  [768] = "0.00,0.00,0.00,90.00,0.00,90.00,0,"
  [769] = "0.00,0.00,0.00,90.00,0.00,90.00,0,"
  [770] = "0.00,0.00,0.00,90.00,0.00,90.00,0,"
  [771] = "0.00,0.00,0.00,90.00,0.00,90.00,1,"
  [772] = "0.00,0.00,0.00,90.00,0.00,90.00,0,"
  [773] = "0.00,0.00,0.00,90.00,0.00,90.00,0,"
  [774] = "0.00,0.00,0.00,90.00,0.00,90.00,0,"
  [775] = "0.00,0.00,0.00,90.00,0.00,90.00,1,"
  [776] = "0.00,0.00,0.00,90.00,0.00,90.00,0,"
  [777] = "0.00,0.00,0.00,90.00,0.00,90.00,0,"
  [778] = "0.00,0.00,0.00,90.00,0.00,90.00,0,"
  [779] = "0.00,0.00,0.00,90.00,0.00,90.00,1,"
  [780] = "0.00,0.00,0.00,90.00,0.00,90.00,0,"
  [781] = "0.00,0.00,0.00,90.00,0.00,90.00,0,"
  [782] = "0.00,0.00,0.00,90.00,0.00,90.00,0,"
  [783] = "0.00,0.00,0.00,90.00,0.00,90.00,1,"
  [784] = "0.00,0.00,0.00,90.00,0.00,90.00,0,"
  [785] = "0.00,0.00,0.00,90.00,0.00,90.00,0,"
  [786] = "0.00,0.00,0.00,90.00,0.00,90.00,0,"
  [787] = "0.00,0.00,0.00,90.00,0.00,90.00,1,"
  [788] = "0.00,0.00,0.00,90.00,0.00,90.00,0,"
  [789] = "0.00,0.00,0.00,90.00,0.00,90.00,0,"
  [790] = "0.00,0.00,0.00,90.00,0.00,90.00,0,"
  [791] = "0.00,0.00,0.00,90.00,0.00,90.00,1,"
  [792] = "0.00,0.00,0.00,90.00,0.00,90.00,0,"
  [793] = "0.00,0.00,0.00,90.00,0.00,90.00,0,"
  [794] = "0.00,0.00,0.00,90.00,0.00,90.00,0,"
  [795] = "0.00,0.00,0.00,90.00,0.00,90.00,1,"
  [796] = "0.00,0.00,0.00,90.00,0.00,90.00,0,"
  [797] = "0.00,0.00,0.00,90.00,0.00,90.00,0,"
  [798] = "0.00,0.00,0.00,90.00,0.00,90.00,0,"
  [799] = "0.00,0.00,0.00,90.00,0.00,90.00,1,"
  [800] = "0.00,0.00,0.00,90.00,0.00,90.00,0,"
  [801] = "0.00,0.00,0.00,90.00,0.00,90.00,0,"
  [802] = "0.00,0.00,0.00,90.00,0.00,90.00,0,"
  [803] = "0.00,0.00,0.00,90.00,0.00,90.00,1,"
  [804] = "0.00,0.00,0.00,90.00,0.00,90.00,0,"
  [805] = "0.00,0.00,0.00,90.00,0.00,90.00,0,"
  [806] = "0.00,0.00,0.00,90.00,0.00,90.00,0,"
  [807] = "0.00,0.00,0.00,90.00,0.00,90.00,1,"
  [808] = "0.00,0.00,0.00,90.00,0.00,90.00,0,"
  [809] = "0.00,0.00,0.00,90.00,0.00,90.00,0,"
  [810] = "0.00,0.00,0.00,90.00,0.00,90.00,0,"
  [811] = "0.00,0.00,0.00,90.00,0.00,90.00,1,"
  [812] = "0.00,0.00,0.00,90.00,0.00,90.00,0,"
  [813] = "0.00,0.00,0.00,90.00,0.00,90.00,0,"
  [814] = "0.00,0.00,0.00,90.00,0.00,90.00,0,"
  [815] = "0.00,0.00,0.00,90.00,0.00,90.00,1,"
  [816] = "0.00,0.00,0.00,90.00,0.00,90.00,0,"
  [817] = "0.00,0.00,0.00,90.00,0.00,90.00,0,"
  [818] = "0.00,0.00,0.00,90.00,0.00,90.00,0,"
  [819] = "0.00,0.00,0.00,90.00,0.00,90.00,1,"
  [820] = "0.00,0.00,0.00,90.00,0.00,90.00,0,"
  [821] = "0.00,0.00,0.00,90.00,0.00,90.00,0,"
  [822] = "0.00,0.00,0.00,90.00,0.00,90.00,0,"
  [823] = "0.00,0.00,0.00,90.00,0.00,90.00,1,"
  [824] = "0.00,0.00,0.00,90.00,0.00,90.00,0,"
  [825] = "0.00,0.00,0.00,90.00,0.00,90.00,0,"
  [826] = "0.00,0.00,0.00,90.00,0.00,90.00,0,"
  [827] = "0.00,0.00,0.00,90.00,0.00,90.00,1,"
  [828] = "0.00,0.00,0.00,90.00,0.00,90.00,0,"
  [829] = "0.00,0.00,0.00,90.00,0.00,90.00,0,"
  [830] = "0.00,0.00,0.00,90.00,0.00,90.00,0,"
  [831] = "0.00,0.00,0.00,90.00,0.00,90.00,1,"
  [832] = "0.00,0.00,0.00,90.00,0.00,90.00,0,"
  [833] = "0.00,0.00,0.00,90.00,0.00,90.00,0,"
  [834] = "0.00,0.00,0.00,90.00,0.00,90.00,0,"
  [835] = "0.00,0.00,0.00,90.00,0.00,90.00,1,"
  [836] = "0.00,0.00,0.00,90.00,0.00,90.00,0,"
  [837] = "0.00,0.00,0.00,90.00,0.00,90.00,0,"
  [838] = "0.00,0.00,0.00,90.00,0.00,90.00,0,"
  [839] = "0.00,0.00,0.00,90.00,0.00,90.00,1,"
  [840] = "0.00,0.00,0.00,90.00,0.00,90.00,0,"
  [841] = "0.00,0.00,0.00,90.00,0.00,90.00,0,"
  [842] = "0.00,0.00,0.00,90.00,0.00,90.00,0,"
  [843] = "0.00,0.00,0.00,90.00,0.00,90.00,1,"
  [844] = "0.00,0.00,0.00,90.00,0.00,90.00,0,"
  [845] = "0.00,0.00,0.00,90.00,0.00,90.00,0,"
  [846] = "0.00,0.00,0.00,90.00,0.00,90.00,0,"
  [847] = "0.00,0.00,0.00,90.00,0.00,90.00,1,"
  [848] = "0.00,0.00,0.00,90.00,0.00,90.00,0,"
  [849] = "0.00,0.00,0.00,90.00,0.00,90.00,0,"
  [850] = "0.00,0.00,0.00,90.00,0.00,90.00,0,"
  [851] = "0.00,0.00,0.00,90.00,0.00,90.00,1,"
  [852] = "0.00,0.00,0.00,90.00,0.00,90.00,0,"
  [853] = "0.00,0.00,0.00,90.00,0.00,90.00,0,"
  [854] = "0.00,0.00,0.00,90.00,0.00,90.00,0,"
  [855] = "0.00,0.00,0.00,90.00,0.00,90.00,1,"
  [856] = "0.00,0.00,0.00,90.00,0.00,90.00,0,"
  [857] = "0.00,0.00,0.00,90.00,0.00,90.00,0,"
  [858] = "0.00,0.00,0.00,90.00,0.00,90.00,0,"
  [859] = "0.00,0.00,0.00,90.00,0.00,90.00,1,"
  [860] = "0.00,0.00,0.00,90.00,0.00,90.00,0,"
  [861] = "0.00,0.00,0.00,90.00,0.00,90.00,0,"
  [862] = "0.00,0.00,0.00,90.00,0.00,90.00,0,"
  [863] = "0.00,0.00,0.00,90.00,0.00,90.00,1,"
  [864] = "0.00,0.00,0.00,90.00,0.00,90.00,0,"
  [865] = "0.00,0.00,0.00,90.00,0.00,90.00,0,"
  [866] = "0.00,0.00,0.00,90.00,0.00,90.00,0,"
  [867] = "0.00,0.00,0.00,90.00,0.00,90.00,1,"
  [868] = "0.00,0.00,0.00,90.00,0.00,90.00,0,"
  [869] = "0.00,0.00,0.00,90.00,0.00,90.00,0,"
  [870] = "0.00,0.00,0.00,90.00,0.00,90.00,0,"
  [871] = "0.00,0.00,0.00,90.00,0.00,90.00,1,"
  [872] = "0.00,0.00,0.00,90.00,0.00,90.00,0,"
  [873] = "0.00,0.00,0.00,90.00,0.00,90.00,0,"
  [874] = "0.00,0.00,0.00,90.00,0.00,90.00,0,"
  [875] = "0.00,0.00,0.00,90.00,0.00,90.00,1,"
  [876] = "0.00,0.00,0.00,90.00,0.00,90.00,0,"
  [877] = "0.00,0.00,0.00,90.00,0.00,90.00,0,"
  [878] = "0.00,0.00,0.00,90.00,0.00,90.00,0,"
  [879] = "0.00,0.00,0.00,90.00,0.00,90.00,1,"
  [880] = "0.00,0.00,0.00,90.00,0.00,90.00,0,"
  [881] = "0.00,0.00,0.00,90.00,0.00,90.00,0,"
  [882] = "0.00,0.00,0.00,90.00,0.00,90.00,0,"
  [883] = "0.00,0.00,0.00,90.00,0.00,90.00,1,"
  [884] = "0.00,0.00,0.00,90.00,0.00,90.00,0,"
  [885] = "0.00,0.00,0.00,90.00,0.00,90.00,0,"
  [886] = "0.00,0.00,0.00,90.00,0.00,90.00,0,"
  [887] = "0.00,0.00,0.00,90.00,0.00,90.00,1,"
  [888] = "0.00,0.00,0.00,90.00,0.00,90.00,0,"
  [889] = "0.00,0.00,0.00,90.00,0.00,90.00,0,"
  [890] = "0.00,0.00,0.00,90.00,0.00,90.00,0,"
  [891] = "0.00,0.00,0.00,90.00,0.00,90.00,1,"
  [892] = "0.00,0.00,0.00,90.00,0.00,90.00,0,"
  [893] = "0.00,0.00,0.00,90.00,0.00,90.00,0,"
  [894] = "0.00,0.00,0.00,90.00,0.00,90.00,0,"
  [895] = "0.00,0.00,0.00,90.00,0.00,90.00,1,"
  [896] = "0.00,0.00,0.00,90.00,0.00,90.00,0,"
  [897] = "0.00,0.00,0.00,90.00,0.00,90.00,0,"
  [898] = "0.00,0.00,0.00,90.00,0.00,90.00,0,"
  [899] = "0.00,0.00,0.00,90.00,0.00,90.00,1,"
  [900] = "0.00,0.00,0.00,90.00,0.00,90.00,0,"
  [901] = "0.00,0.00,0.00,90.00,0.00,90.00,0,"
  [902] = "0.00,0.00,0.00,90.00,0.00,90.00,0,"
  [903] = "0.00,0.00,0.00,90.00,0.00,90.00,1,"
  [904] = "0.00,0.00,0.00,90.00,0.00,90.00,0,"
  [905] = "0.00,0.00,0.00,90.00,0.00,90.00,0,"
  [906] = "0.00,0.00,0.00,90.00,0.00,90.00,0,"
  [907] = "0.00,0.00,0.00,90.00,0.00,90.00,1,"
  [908] = "0.00,0.00,0.00,90.00,0.00,90.00,0,"
  [909] = "0.00,0.00,0.00,90.00,0.00,90.00,0,"
  [910] = "0.00,0.00,0.00,90.00,0.00,90.00,0,"
  [911] = "0.00,0.00,0.00,90.00,0.00,90.00,1,"
  [912] = "0.00,0.00,0.00,90.00,0.00,90.00,0,"
  [913] = "0.00,0.00,0.00,90.00,0.00,90.00,0,"
  [914] = "0.00,0.00,0.00,90.00,0.00,90.00,0,"
  [915] = "0.00,0.00,0.00,90.00,0.00,90.00,1,"
  [916] = "0.00,0.00,0.00,90.00,0.00,90.00,0,"
  [917] = "0.00,0.00,0.00,90.00,0.00,90.00,0,"
  [918] = "0.00,0.00,0.00,90.00,0.00,90.00,0,"
  [919] = "0.00,0.00,0.00,90.00,0.00,90.00,1,"
  [920] = "0.00,0.00,0.00,90.00,0.00,90.00,0,"
  [921] = "0.00,0.00,0.00,90.00,0.00,90.00,0,"
  [922] = "0.00,0.00,0.00,90.00,0.00,90.00,0,"
  [923] = "0.00,0.00,0.00,90.00,0.00,90.00,1,"
  [924] = "0.00,0.00,0.00,90.00,0.00,90.00,0,"
  [925] = "0.00,0.00,0.00,90.00,0.00,90.00,0,"
  [926] = "0.00,0.00,0.00,90.00,0.00,90.00,0,"
  [927] = "0.00,0.00,0.00,90.00,0.00,90.00,1,"
  [928] = "0.00,0.00,0.00,90.00,0.00,90.00,0,"
  [929] = "0.00,0.00,0.00,90.00,0.00,90.00,0,"
  [930] = "0.00,0.00,0.00,90.00,0.00,90.00,0,"
  [931] = "0.00,0.00,0.00,90.00,0.00,90.00,1,"
  [932] = "0.00,0.00,0.00,90.00,0.00,90.00,0,"
  [933] = "0.00,0.00,0.00,90.00,0.00,90.00,0,"
  [934] = "0.00,0.00,0.00,90.00,0.00,90.00,0,"
  [935] = "0.00,0.00,0.00,90.00,0.00,90.00,1,"
  [936] = "0.00,0.00,0.00,90.00,0.00,90.00,0,"
  [937] = "0.00,0.00,0.00,90.00,0.00,90.00,0,"
  [938] = "0.00,0.00,0.00,90.00,0.00,90.00,0,"
  [939] = "0.00,0.00,0.00,90.00,0.00,90.00,1,"
  [940] = "0.00,0.00,0.00,90.00,0.00,90.00,0,"
  [941] = "0.00,0.00,0.00,90.00,0.00,90.00,0,"
  [942] = "0.00,0.00,0.00,90.00,0.00,90.00,0,"
  [943] = "0.00,0.00,0.00,90.00,0.00,90.00,1,"
  [944] = "0.00,0.00,0.00,90.00,0.00,90.00,0,"
  [945] = "0.00,0.00,0.00,90.00,0.00,90.00,0,"
  [946] = "0.00,0.00,0.00,90.00,0.00,90.00,0,"
  [947] = "0.00,0.00,0.00,90.00,0.00,90.00,1,"
  [948] = "0.00,0.00,0.00,90.00,0.00,90.00,0,"
  [949] = "0.00,0.00,0.00,90.00,0.00,90.00,0,"
  [950] = "0.00,0.00,0.00,90.00,0.00,90.00,0,"
  [951] = "0.00,0.00,0.00,90.00,0.00,90.00,1,"
  [952] = "0.00,0.00,0.00,90.00,0.00,90.00,0,"
  [953] = "0.00,0.00,0.00,90.00,0.00,90.00,0,"
  [954] = "0.00,0.00,0.00,90.00,0.00,90.00,0,"
  [955] = "0.00,0.00,0.00,90.00,0.00,90.00,1,"
  [956] = "0.00,0.00,0.00,90.00,0.00,90.00,0,"
  [957] = "0.00,0.00,0.00,90.00,0.00,90.00,0,"
  [958] = "0.00,0.00,0.00,90.00,0.00,90.00,0,"
  [959] = "0.00,0.00,0.00,90.00,0.00,90.00,1,"
  [960] = "0.00,0.00,0.00,90.00,0.00,90.00,0,"
  [961] = "0.00,0.00,0.00,90.00,0.00,90.00,0,"
  [962] = "0.00,0.00,0.00,90.00,0.00,90.00,0,"
  [963] = "0.00,0.00,0.00,90.00,0.00,90.00,1,"
  [964] = "0.00,0.00,0.00,90.00,0.00,90.00,0,"
  [965] = "0.00,0.00,0.00,90.00,0.00,90.00,0,"
  [966] = "0.00,0.00,0.00,90.00,0.00,90.00,0,"
  [967] = "0.00,0.00,0.00,90.00,0.00,90.00,1,"
  [968] = "0.00,0.00,0.00,90.00,0.00,90.00,0,"
  [969] = "0.00,0.00,0.00,90.00,0.00,90.00,0,"
  [970] = "0.00,0.00,0.00,90.00,0.00,90.00,0,"
  [971] = "0.00,0.00,0.00,90.00,0.00,90.00,1,"
  [972] = "0.00,0.00,0.00,90.00,0.00,90.00,0,"
  [973] = "0.00,0.00,0.00,90.00,0.00,90.00,0,"
  [974] = "0.00,0.00,0.00,90.00,0.00,90.00,0,"
  [975] = "0.00,0.00,0.00,90.00,0.00,90.00,1,"
  [976] = "0.00,0.00,0.00,90.00,0.00,90.00,0,"
  [977] = "0.00,0.00,0.00,90.00,0.00,90.00,0,"
  [978] = "0.00,0.00,0.00,90.00,0.00,90.00,0,"
  [979] = "0.00,0.00,0.00,90.00,0.00,90.00,1,"
  [980] = "0.00,0.00,0.00,90.00,0.00,90.00,0,"
  [981] = "0.00,0.00,0.00,90.00,0.00,90.00,0,"
  [982] = "0.00,0.00,0.00,90.00,0.00,90.00,0,"
  [983] = "0.00,0.00,0.00,90.00,0.00,90.00,1,"
  [984] = "0.00,0.00,0.00,90.00,0.00,90.00,0,"
  [985] = "0.00,0.00,0.00,90.00,0.00,90.00,0,"
  [986] = "0.00,0.00,0.00,90.00,0.00,90.00,0,"
  [987] = "0.00,0.00,0.00,90.00,0.00,90.00,1,"
  [988] = "0.00,0.00,0.00,90.00,0.00,90.00,0,"
  [989] = "0.00,0.00,0.00,90.00,0.00,90.00,0,"
  [990] = "0.00,0.00,0.00,90.00,0.00,90.00,0,"
  [991] = "0.00,0.00,0.00,90.00,0.00,90.00,1,"
  [992] = "0.00,0.00,0.00,90.00,0.00,90.00,0,"
  [993] = "0.00,0.00,0.00,90.00,0.00,90.00,0,"
  [994] = "0.00,0.00,0.00,90.00,0.00,90.00,0,"
  [995] = "0.00,0.00,0.00,90.00,0.00,90.00,1,"
  [996] = "0.00,0.00,0.00,90.00,0.00,90.00,0,"
  [997] = "0.00,0.00,0.00,90.00,0.00,90.00,0,"
  [998] = "0.00,0.00,0.00,90.00,0.00,90.00,0,"
  [999] = "0.00,0.00,0.00,90.00,0.00,90.00,1,"
  [1000] = "0.00,0.00,0.00,90.00,0.00,90.00,0,"
  [1001] = "0.00,0.00,0.00,90.00,0.00,90.00,0,"
  [1002] = "0.00,0.00,0.00,90.00,0.00,90.00,0,"
  [1003] = "0.00,0.00,0.00,90.00,0.00,90.00,1,"
  [1004] = "0.00,0.00,0.00,90.00,0.00,90.00,0,"
  [1005] = "0.00,0.00,0.00,90.00,0.00,90.00,0,"
  [1006] = "0.00,0.00,0.00,90.00,0.00,90.00,0,"
  [1007] = "0.00,0.00,0.00,90.00,0.00,90.00,1,"
  [1008] = "0.00,0.00,0.00,90.00,0.00,90.00,0,"
  [1009] = "0.00,0.00,0.00,90.00,0.00,90.00,0,"
  [1010] = "0.00,0.00,0.00,90.00,0.00,90.00,0,"
  [1011] = "0.00,0.00,0.00,90.00,0.00,90.00,1,"
  [1012] = "0.00,0.00,0.00,90.00,0.00,90.00,0,"
  [1013] = "0.00,0.00,0.00,90.00,0.00,90.00,0,"
  [1014] = "0.00,0.00,0.00,90.00,0.00,90.00,0,"
  [1015] = "0.00,0.00,0.00,90.00,0.00,90.00,1,"
  [1016] = "0.00,0.00,0.00,90.00,0.00,90.00,0,"
  [1017] = "0.00,0.00,0.00,90.00,0.00,90.00,0,"
  [1018] = "0.00,0.00,0.00,90.00,0.00,90.00,0,"
  [1019] = "0.00,0.00,0.00,90.00,0.00,90.00,1,"
  [1020] = "0.00,0.00,0.00,90.00,0.00,90.00,0,"
  [1021] = "0.00,0.00,0.00,90.00,0.00,90.00,0,"
  [1022] = "0.00,0.00,0.00,90.00,0.00,90.00,0,"
  [1023] = "0.00,0.00,0.00,90.00,0.00,90.00,1,"
  [1024] = "0.00,0.00,0.00,90.00,0.00,90.00,0,"
  [1025] = "0.00,0.00,0.00,90.00,0.00,90.00,0,"
  [1026] = "0.00,0.00,0.00,90.00,0.00,90.00,0,"
  [1027] = "0.00,0.00,0.00,90.00,0.00,90.00,1,"
  [1028] = "0.00,0.00,0.00,90.00,0.00,90.00,0,"
  [1029] = "0.00,0.00,0.00,90.00,0.00,90.00,0,"
  [1030] = "0.00,0.00,0.00,90.00,0.00,90.00,0,"
  [1031] = "0.00,0.00,0.00,90.00,0.00,90.00,1,"
  [1032] = "0.00,0.00,0.00,90.00,0.00,90.00,0,"
  [1033] = "0.00,0.00,0.00,90.00,0.00,90.00,0,"
  [1034] = "0.00,0.00,0.00,90.00,0.00,90.00,0,"
  [1035] = "0.00,0.00,0.00,90.00,0.00,90.00,1,"
  [1036] = "0.00,0.00,0.00,90.00,0.00,90.00,0,"
  [1037] = "0.00,0.00,0.00,90.00,0.00,90.00,0,"
  [1038] = "0.00,0.00,0.00,90.00,0.00,90.00,0,"
  [1039] = "0.00,0.00,0.00,90.00,0.00,90.00,1,"
  [1040] = "0.00,0.00,0.00,90.00,0.00,90.00,0,"
  [1041] = "0.00,0.00,0.00,90.00,0.00,90.00,0,"
  [1042] = "0.00,0.00,0.00,90.00,0.00,90.00,0,"
  [1043] = "0.00,0.00,0.00,90.00,0.00,90.00,1,"
  [1044] = "0.00,0.00,0.00,90.00,0.00,90.00,0,"
  [1045] = "0.00,0.00,0.00,90.00,0.00,90.00,0,"
  [1046] = "0.00,0.00,0.00,90.00,0.00,90.00,0,"
  [1047] = "0.00,0.00,0.00,90.00,0.00,90.00,1,"
  [1048] = "0.00,0.00,0.00,90.00,0.00,90.00,0,"
  [1049] = "0.00,0.00,0.00,90.00,0.00,90.00,0,"
  [1050] = "0.00,0.00,0.00,90.00,0.00,90.00,0,"
  [1051] = "0.00,0.00,0.00,90.00,0.00,90.00,1,"
  [1052] = "0.00,0.00,0.00,90.00,0.00,90.00,0,"
  [1053] = "0.00,0.00,0.00,90.00,0.00,90.00,0,"
  [1054] = "0.00,0.00,0.00,90.00,0.00,90.00,0,"
  [1055] = "0.00,0.00,0.00,90.00,0.00,90.00,1,"
  [1056] = "0.00,0.00,0.00,90.00,0.00,90.00,0,"
  [1057] = "0.00,0.00,0.00,90.00,0.00,90.00,0,"
  [1058] = "0.00,0.00,0.00,90.00,0.00,90.00,0,"
  [1059] = "0.00,0.00,0.00,90.00,0.00,90.00,1,"
  [1060] = "0.00,0.00,0.00,90.00,0.00,90.00,0,"
  [1061] = "0.00,0.00,0.00,90.00,0.00,90.00,0,"
  [1062] = "0.00,0.00,0.00,90.00,0.00,90.00,0,"
  [1063] = "0.00,0.00,0.00,90.00,0.00,90.00,1,"
  [1064] = "0.00,0.00,0.00,90.00,0.00,90.00,0,"
  [1065] = "0.00,0.00,0.00,90.00,0.00,90.00,0,"
  [1066] = "0.00,0.00,0.00,90.00,0.00,90.00,0,"
  [1067] = "0.00,0.00,0.00,90.00,0.00,90.00,1,"
  [1068] = "0.00,0.00,0.00,90.00,0.00,90.00,0,"
  [1069] = "0.00,0.00,0.00,90.00,0.00,90.00,0,"
  [1070] = "0.00,0.00,0.00,90.00,0.00,90.00,0,"
  [1071] = "0.00,0.00,0.00,90.00,0.00,90.00,1,"
  [1072] = "0.00,0.00,0.00,90.00,0.00,90.00,0,"
  [1073] = "0.00,0.00,0.00,90.00,0.00,90.00,0,"
  [1074] = "0.00,0.00,0.00,90.00,0.00,90.00,0,"
  [1075] = "0.00,0.00,0.00,90.00,0.00,90.00,1,"
  [1076] = "0.00,0.00,0.00,90.00,0.00,90.00,0,"
  [1077] = "0.00,0.00,0.00,90.00,0.00,90.00,0,"
  [1078] = "0.00,0.00,0.00,90.00,0.00,90.00,0,"
  [1079] = "0.00,0.00,0.00,90.00,0.00,90.00,1,"
  [1080] = "0.00,0.00,0.00,90.00,0.00,90.00,0,"
  [1081] = "0.00,0.00,0.00,90.00,0.00,90.00,0,"
  [1082] = "0.00,0.00,0.00,90.00,0.00,90.00,0,"
  [1083] = "0.00,0.00,0.00,90.00,0.00,90.00,1,"
  [1084] = "0.00,0.00,0.00,90.00,0.00,90.00,0,"
  [1085] = "0.00,0.00,0.00,90.00,0.00,90.00,0,"
  [1086] = "0.00,0.00,0.00,90.00,0.00,90.00,0,"
  [1087] = "0.00,0.00,0.00,90.00,0.00,90.00,1,"
  [1088] = "0.00,0.00,0.00,90.00,0.00,90.00,0,"
  [1089] = "0.00,0.00,0.00,90.00,0.00,90.00,0,"
  [1090] = "0.00,0.00,0.00,90.00,0.00,90.00,0,"
  [1091] = "0.00,0.00,0.00,90.00,0.00,90.00,1,"
  [1092] = "0.00,0.00,0.00,90.00,0.00,90.00,0,"
  [1093] = "0.00,0.00,0.00,90.00,0.00,90.00,0,"
  [1094] = "0.00,0.00,0.00,90.00,0.00,90.00,0,"
  [1095] = "0.00,0.00,0.00,90.00,0.00,90.00,1,"
  [1096] = "0.00,0.00,0.00,90.00,0.00,90.00,0,"
  [1097] = "0.00,0.00,0.00,90.00,0.00,90.00,0,"
  [1098] = "0.00,0.00,0.00,90.00,0.00,90.00,0,"
  [1099] = "0.00,0.00,0.00,90.00,0.00,90.00,1,"
  [1100] = "0.00,0.00,0.00,90.00,0.00,90.00,0,"
  [1101] = "0.00,0.00,0.00,90.00,0.00,90.00,0,"
  [1102] = "0.00,0.00,0.00,90.00,0.00,90.00,0,"
  [1103] = "0.00,0.00,0.00,90.00,0.00,90.00,1,"
  [1104] = "0.00,0.00,0.00,90.00,0.00,90.00,0,"
  [1105] = "0.00,0.00,0.00,90.00,0.00,90.00,0,"
  [1106] = "0.00,0.00,0.00,90.00,0.00,90.00,0,"
  [1107] = "0.00,0.00,0.00,90.00,0.00,90.00,1,"
  [1108] = "0.00,0.00,0.00,90.00,0.00,90.00,0,"
  [1109] = "0.00,0.00,0.00,90.00,0.00,90.00,0,"
  [1110] = "0.00,0.00,0.00,90.00,0.00,90.00,0,"
  [1111] = "0.00,0.00,0.00,90.00,0.00,90.00,1,"
  [1112] = "0.00,0.00,0.00,90.00,0.00,90.00,0,"
  [1113] = "0.00,0.00,0.00,90.00,0.00,90.00,0,"
  [1114] = "0.00,0.00,0.00,90.00,0.00,90.00,0,"
  [1115] = "0.00,0.00,0.00,90.00,0.00,90.00,1,"
  [1116] = "0.00,0.00,0.00,90.00,0.00,90.00,0,"
  [1117] = "0.00,0.00,0.00,90.00,0.00,90.00,0,"
  [1118] = "0.00,0.00,0.00,90.00,0.00,90.00,0,"
  [1119] = "0.00,0.00,0.00,90.00,0.00,90.00,1,"
  [1120] = "0.00,0.00,0.00,90.00,0.00,90.00,0,"
  [1121] = "0.00,0.00,0.00,90.00,0.00,90.00,0,"
  [1122] = "0.00,0.00,0.00,90.00,0.00,90.00,0,"
  [1123] = "0.00,0.00,0.00,90.00,0.00,90.00,1,"
  [1124] = "0.00,0.00,0.00,90.00,0.00,90.00,0,"
  [1125] = "0.00,0.00,0.00,90.00,0.00,90.00,0,"
  [1126] = "0.00,0.00,0.00,90.00,0.00,90.00,0,"
  [1127] = "0.00,0.00,0.00,90.00,0.00,90.00,1,"
  [1128] = "0.00,0.00,0.00,90.00,0.00,90.00,0,"
  [1129] = "0.00,0.00,0.00,90.00,0.00,90.00,0,"
  [1130] = "0.00,0.00,0.00,90.00,0.00,90.00,0,"
  [1131] = "0.00,0.00,0.00,90.00,0.00,90.00,1,"
  [1132] = "0.00,0.00,0.00,90.00,0.00,90.00,0,"
  [1133] = "0.00,0.00,0.00,90.00,0.00,90.00,0,"
  [1134] = "0.00,0.00,0.00,90.00,0.00,90.00,0,"
  [1135] = "0.00,0.00,0.00,90.00,0.00,90.00,1,"
  [1136] = "0.00,0.00,0.00,90.00,0.00,90.00,0,"
  [1137] = "0.00,0.00,0.00,90.00,0.00,90.00,0,"
  [1138] = "0.00,0.00,0.00,90.00,0.00,90.00,0,"
  [1139] = "0.00,0.00,0.00,90.00,0.00,90.00,1,"
  [1140] = "0.00,0.00,0.00,90.00,0.00,90.00,0,"
  [1141] = "0.00,0.00,0.00,90.00,0.00,90.00,0,"
  [1142] = "0.00,0.00,0.00,90.00,0.00,90.00,0,"
  [1143] = "0.00,0.00,0.00,90.00,0.00,90.00,1,"
  [1144] = "0.00,0.00,0.00,90.00,0.00,90.00,0,"
  [1145] = "0.00,0.00,0.00,90.00,0.00,90.00,0,"
  [1146] = "0.00,0.00,0.00,90.00,0.00,90.00,0,"
  [1147] = "0.00,0.00,0.00,90.00,0.00,90.00,1,"
  [1148] = "0.00,0.00,0.00,90.00,0.00,90.00,0,"
  [1149] = "0.00,0.00,0.00,90.00,0.00,90.00,0,"
  [1150] = "0.00,0.00,0.00,90.00,0.00,90.00,0,"
  [1151] = "0.00,0.00,0.00,90.00,0.00,90.00,1,"
  [1152] = "0.00,0.00,0.00,90.00,0.00,90.00,0,"
  [1153] = "0.00,0.00,0.00,90.00,0.00,90.00,0,"
  [1154] = "0.00,0.00,0.00,90.00,0.00,90.00,0,"
  [1155] = "0.00,0.00,0.00,90.00,0.00,90.00,1,"
  [1156] = "0.00,0.00,0.00,90.00,0.00,90.00,0,"
  [1157] = "0.00,0.00,0.00,90.00,0.00,90.00,0,"
  [1158] = "0.00,0.00,0.00,90.00,0.00,90.00,0,"
  [1159] = "0.00,0.00,0.00,90.00,0.00,90.00,1,"
  [1160] = "0.00,0.00,0.00,90.00,0.00,90.00,0,"
  [1161] = "0.00,0.00,0.00,90.00,0.00,90.00,0,"
  [1162] = "0.00,0.00,0.00,90.00,0.00,90.00,0,"
  [1163] = "0.00,0.00,0.00,90.00,0.00,90.00,1,"
  [1164] = "0.00,0.00,0.00,90.00,0.00,90.00,0,"
  [1165] = "0.00,0.00,0.00,90.00,0.00,90.00,0,"
  [1166] = "0.00,0.00,0.00,90.00,0.00,90.00,0,"
  [1167] = "0.00,0.00,0.00,90.00,0.00,90.00,1,"
  [1168] = "0.00,0.00,0.00,90.00,0.00,90.00,0,"
  [1169] = "0.00,0.00,0.00,90.00,0.00,90.00,0,"
  [1170] = "0.00,0.00,0.00,90.00,0.00,90.00,0,"
  [1171] = "0.00,0.00,0.00,90.00,0.00,90.00,1,"
  [1172] = "0.00,0.00,0.00,90.00,0.00,90.00,0,"
  [1173] = "0.00,0.00,0.00,90.00,0.00,90.00,0,"
  [1174] = "0.00,0.00,0.00,90.00,0.00,90.00,0,"
  [1175] = "0.00,0.00,0.00,90.00,0.00,90.00,1,"
  [1176] = "0.00,0.00,0.00,90.00,0.00,90.00,0,"
  [1177] = "0.00,0.00,0.00,90.00,0.00,90.00,0,"
  [1178] = "0.00,0.00,0.00,90.00,0.00,90.00,0,"
  [1179] = "0.00,0.00,0.00,90.00,0.00,90.00,1,"
  [1180] = "0.00,0.00,0.00,90.00,0.00,90.00,0,"
  [1181] = "0.00,0.00,0.00,90.00,0.00,90.00,0,"
  [1182] = "0.00,0.00,0.00,90.00,0.00,90.00,0,"
  [1183] = "0.00,0.00,0.00,90.00,0.00,90.00,1,"
  [1184] = "0.00,0.00,0.00,90.00,0.00,90.00,0,"
  [1185] = "0.00,0.00,0.00,90.00,0.00,90.00,0,"
  [1186] = "0.00,0.00,0.00,90.00,0.00,90.00,0,"
  [1187] = "0.00,0.00,0.00,90.00,0.00,90.00,1,"
  [1188] = "0.00,0.00,0.00,90.00,0.00,90.00,0,"
  [1189] = "0.00,0.00,0.00,90.00,0.00,90.00,0,"
  [1190] = "0.00,0.00,0.00,90.00,0.00,90.00,0,"
  [1191] = "0.00,0.00,0.00,90.00,0.00,90.00,1,"
  [1192] = "0.00,0.00,0.00,90.00,0.00,90.00,0,"
  [1193] = "0.00,0.00,0.00,90.00,0.00,90.00,0,"
  [1194] = "0.00,0.00,0.00,90.00,0.00,90.00,0,"
  [1195] = "0.00,0.00,0.00,90.00,0.00,90.00,1,"
  [1196] = "0.00,0.00,0.00,90.00,0.00,90.00,0,"
  [1197] = "0.00,0.00,0.00,90.00,0.00,90.00,0,"
  [1198] = "0.00,0.00,0.00,90.00,0.00,90.00,0,"
  [1199] = "0.00,0.00,0.00,90.00,0.00,90.00,1,"
  [1200] = "0.00,0.00,0.00,90.00,0.00,90.00,0,"
  [1201] = "0.00,0.00,0.00,90.00,0.00,90.00,0,"
  [1202] = "0.00,0.00,0.00,90.00,0.00,90.00,0,"
  [1203] = "0.00,0.00,0.00,90.00,0.00,90.00,1,"
  [1204] = "0.00,0.00,0.00,90.00,0.00,90.00,0,"
  [1205] = "0.00,0.00,0.00,90.00,0.00,90.00,0,"
  [1206] = "0.00,0.00,0.00,90.00,0.00,90.00,0,"
  [1207] = "0.00,0.00,0.00,90.00,0.00,90.00,1,"
  [1208] = "0.00,0.00,0.00,90.00,0.00,90.00,0,"
  [1209] = "0.00,0.00,0.00,90.00,0.00,90.00,0,"
  [1210] = "0.00,0.00,0.00,90.00,0.00,90.00,0,"
  [1211] = "0.00,0.00,0.00,90.00,0.00,90.00,1,"
  [1212] = "0.00,0.00,0.00,90.00,0.00,90.00,0,"
  [1213] = "0.00,0.00,0.00,90.00,0.00,90.00,0,"
  [1214] = "0.00,0.00,0.00,90.00,0.00,90.00,0,"
  [1215] = "0.00,0.00,0.00,90.00,0.00,90.00,1,"
  [1216] = "0.00,0.00,0.00,90.00,0.00,90.00,0,"
  [1217] = "0.00,0.00,0.00,90.00,0.00,90.00,0,"
  [1218] = "0.00,0.00,0.00,90.00,0.00,90.00,0,"
  [1219] = "0.00,0.00,0.00,90.00,0.00,90.00,1,"
  [1220] = "0.00,0.00,0.00,90.00,0.00,90.00,0,"
  [1221] = "0.00,0.00,0.00,90.00,0.00,90.00,0,"
  [1222] = "0.00,0.00,0.00,90.00,0.00,90.00,0,"
  [1223] = "0.00,0.00,0.00,90.00,0.00,90.00,1,"
  [1224] = "0.00,0.00,0.00,90.00,0.00,90.00,0,"
  [1225] = "0.00,0.00,0.00,90.00,0.00,90.00,0,"
  [1226] = "0.00,0.00,0.00,90.00,0.00,90.00,0,"
  [1227] = "0.00,0.00,0.00,90.00,0.00,90.00,1,"
  [1228] = "0.00,0.00,0.00,90.00,0.00,90.00,0,"
  [1229] = "0.00,0.00,0.00,90.00,0.00,90.00,0,"
  [1230] = "0.00,0.00,0.00,90.00,0.00,90.00,0,"
  [1231] = "0.00,0.00,0.00,90.00,0.00,90.00,1,"
  [1232] = "0.00,0.00,0.00,90.00,0.00,90.00,0,"
  [1233] = "0.00,0.00,0.00,90.00,0.00,90.00,0,"
  [1234] = "0.00,0.00,0.00,90.00,0.00,90.00,0,"
  [1235] = "0.00,0.00,0.00,90.00,0.00,90.00,1,"
  [1236] = "0.00,0.00,0.00,90.00,0.00,90.00,0,"
  [1237] = "0.00,0.00,0.00,90.00,0.00,90.00,0,"
  [1238] = "0.00,0.00,0.00,90.00,0.00,90.00,0,"
  [1239] = "0.00,0.00,0.00,90.00,0.00,90.00,1,"
  [1240] = "0.00,0.00,0.00,90.00,0.00,90.00,0,"
  [1241] = "0.00,0.00,0.00,90.00,0.00,90.00,0,"
  [1242] = "0.00,0.00,0.00,90.00,0.00,90.00,0,"
  [1243] = "0.00,0.00,0.00,90.00,0.00,90.00,1,"
  [1244] = "0.00,0.00,0.00,90.00,0.00,90.00,0,"
  [1245] = "0.00,0.00,0.00,90.00,0.00,90.00,0,"
  [1246] = "0.00,0.00,0.00,90.00,0.00,90.00,0,"
  [1247] = "0.00,0.00,0.00,90.00,0.00,90.00,1,"
  [1248] = "0.00,0.00,0.00,90.00,0.00,90.00,0,"
  [1249] = "0.00,0.00,0.00,90.00,0.00,90.00,0,"
  [1250] = "0.00,0.00,0.00,90.00,0.00,90.00,0,"
  [1251] = "0.00,0.00,0.00,90.00,0.00,90.00,1,"
  [1252] = "0.00,0.00,0.00,90.00,0.00,90.00,0,"
  [1253] = "0.00,0.00,0.00,90.00,0.00,90.00,0,"
  [1254] = "0.00,0.00,0.00,90.00,0.00,90.00,0,"
  [1255] = "0.00,0.00,0.00,90.00,0.00,90.00,1,"
  [1256] = "0.00,0.00,0.00,90.00,0.00,90.00,0,"
  [1257] = "0.00,0.00,0.00,90.00,0.00,90.00,0,"
  [1258] = "0.00,0.00,0.00,90.00,0.00,90.00,0,"
  [1259] = "0.00,0.00,0.00,90.00,0.00,90.00,1,"
  [1260] = "0.00,0.00,0.00,90.00,0.00,90.00,0,"
  [1261] = "0.00,0.00,0.00,90.00,0.00,90.00,0,"
  [1262] = "0.00,0.00,0.00,90.00,0.00,90.00,0,"
  [1263] = "0.00,0.00,0.00,90.00,0.00,90.00,1,"
  [1264] = "0.00,0.00,0.00,90.00,0.00,90.00,0,"
  [1265] = "0.00,0.00,0.00,90.00,0.00,90.00,0,"
  [1266] = "0.00,0.00,0.00,90.00,0.00,90.00,0,"
  [1267] = "0.00,0.00,0.00,90.00,0.00,90.00,1,"
  [1268] = "0.00,0.00,0.00,90.00,0.00,90.00,0,"
  [1269] = "0.00,0.00,0.00,90.00,0.00,90.00,0,"
  [1270] = "0.00,0.00,0.00,90.00,0.00,90.00,0,"
  [1271] = "0.00,0.00,0.00,90.00,0.00,90.00,1,"
  [1272] = "0.00,0.00,0.00,90.00,0.00,90.00,0,"
  [1273] = "0.00,0.00,0.00,90.00,0.00,90.00,0,"
  [1274] = "0.00,0.00,0.00,90.00,0.00,90.00,0,"
  [1275] = "0.00,0.00,0.00,90.00,0.00,90.00,1,"
  [1276] = "0.00,0.00,0.00,90.00,0.00,90.00,0,"
  [1277] = "0.00,0.00,0.00,90.00,0.00,90.00,0,"
  [1278] = "0.00,0.00,0.00,90.00,0.00,90.00,0,"
  [1279] = "0.00,0.00,0.00,90.00,0.00,90.00,1,"
  [1280] = "0.00,0.00,0.00,90.00,0.00,90.00,0,"
  [1281] = "0.00,0.00,0.00,90.00,0.00,90.00,0,"
  [1282] = "0.00,0.00,0.00,90.00,0.00,90.00,0,"
  [1283] = "0.00,0.00,0.00,90.00,0.00,90.00,1,"
  [1284] = "0.00,0.00,0.00,90.00,0.00,90.00,0,"
  [1285] = "0.00,0.00,0.00,90.00,0.00,90.00,0,"
  [1286] = "0.00,0.00,0.00,90.00,0.00,90.00,0,"
  [1287] = "0.00,0.00,0.00,90.00,0.00,90.00,1,"
  [1288] = "0.00,0.00,0.00,90.00,0.00,90.00,0,"
  [1289] = "0.00,0.00,0.00,90.00,0.00,90.00,0,"
  [1290] = "0.00,0.00,0.00,90.00,0.00,90.00,0,"
  [1291] = "0.00,0.00,0.00,90.00,0.00,90.00,1,"
  [1292] = "0.00,0.00,0.00,90.00,0.00,90.00,0,"
  [1293] = "0.00,0.00,0.00,90.00,0.00,90.00,0,"
  [1294] = "0.00,0.00,0.00,90.00,0.00,90.00,0,"
  [1295] = "0.00,0.00,0.00,90.00,0.00,90.00,1,"
  [1296] = "0.00,0.00,0.00,90.00,0.00,90.00,0,"
  [1297] = "0.00,0.00,0.00,90.00,0.00,90.00,0,"
  [1298] = "0.00,0.00,0.00,90.00,0.00,90.00,0,"
  [1299] = "0.00,0.00,0.00,90.00,0.00,90.00,1,"
  [1300] = "0.00,0.00,0.00,90.00,0.00,90.00,0,"
  [1301] = "0.00,0.00,0.00,90.00,0.00,90.00,0,"
  [1302] = "0.00,0.00,0.00,90.00,0.00,90.00,0,"
  [1303] = "0.00,0.00,0.00,90.00,0.00,90.00,1,"
  [1304] = "0.00,0.00,0.00,90.00,0.00,90.00,0,"
  [1305] = "0.00,0.00,0.00,90.00,0.00,90.00,0,"
  [1306] = "0.00,0.00,0.00,90.00,0.00,90.00,0,"
  [1307] = "0.00,0.00,0.00,90.00,0.00,90.00,1,"
  [1308] = "0.00,0.00,0.00,90.00,0.00,90.00,0,"
  [1309] = "0.00,0.00,0.00,90.00,0.00,90.00,0,"
  [1310] = "0.00,0.00,0.00,90.00,0.00,90.00,0,"
  [1311] = "0.00,0.00,0.00,90.00,0.00,90.00,1,"
  [1312] = "0.00,0.00,0.00,90.00,0.00,90.00,0,"
  [1313] = "0.00,0.00,0.00,90.00,0.00,90.00,0,"
  [1314] = "0.00,0.00,0.00,90.00,0.00,90.00,0,"
  [1315] = "0.00,0.00,0.00,90.00,0.00,90.00,1,"
  [1316] = "0.00,0.00,0.00,90.00,0.00,90.00,0,"
  [1317] = "0.00,0.00,0.00,90.00,0.00,90.00,0,"
  [1318] = "0.00,0.00,0.00,90.00,0.00,90.00,0,"
  [1319] = "0.00,0.00,0.00,90.00,0.00,90.00,1,"
  [1320] = "0.00,0.00,0.00,90.00,0.00,90.00,0,"
  [1321] = "0.00,0.00,0.00,90.00,0.00,90.00,0,"
  [1322] = "0.00,0.00,0.00,90.00,0.00,90.00,0,"
  [1323] = "0.00,0.00,0.00,90.00,0.00,90.00,1,"
  [1324] = "0.00,0.00,0.00,90.00,0.00,90.00,0,"
  [1325] = "0.00,0.00,0.00,90.00,0.00,90.00,0,"
  [1326] = "0.00,0.00,0.00,90.00,0.00,90.00,0,"
  [1327] = "0.00,0.00,0.00,90.00,0.00,90.00,1,"
  [1328] = "0.00,0.00,0.00,90.00,0.00,90.00,0,"
  [1329] = "0.00,0.00,0.00,90.00,0.00,90.00,0,"
  [1330] = "0.00,0.00,0.00,90.00,0.00,90.00,0,"
  [1331] = "0.00,0.00,0.00,90.00,0.00,90.00,1,"
  [1332] = "0.00,0.00,0.00,90.00,0.00,90.00,0,"
  [1333] = "0.00,0.00,0.00,90.00,0.00,90.00,0,"
  [1334] = "0.00,0.00,0.00,90.00,0.00,90.00,0,"
  [1335] = "0.00,0.00,0.00,90.00,0.00,90.00,1,"
  [1336] = "0.00,0.00,0.00,90.00,0.00,90.00,0,"
  [1337] = "0.00,0.00,0.00,90.00,0.00,90.00,0,"
  [1338] = "0.00,0.00,0.00,90.00,0.00,90.00,0,"
  [1339] = "0.00,0.00,0.00,90.00,0.00,90.00,1,"
  [1340] = "0.00,0.00,0.00,90.00,0.00,90.00,0,"
  [1341] = "0.00,0.00,0.00,90.00,0.00,90.00,0,"
  [1342] = "0.00,0.00,0.00,90.00,0.00,90.00,0,"
  [1343] = "0.00,0.00,0.00,90.00,0.00,90.00,1,"
  [1344] = "0.00,0.00,0.00,90.00,0.00,90.00,0,"
  [1345] = "0.00,0.00,0.00,90.00,0.00,90.00,0,"
  [1346] = "0.00,0.00,0.00,90.00,0.00,90.00,0,"
  [1347] = "0.00,0.00,0.00,90.00,0.00,90.00,1,"
  [1348] = "0.00,0.00,0.00,90.00,0.00,90.00,0,"
  [1349] = "0.00,0.00,0.00,90.00,0.00,90.00,0,"
  [1350] = "0.00,0.00,0.00,90.00,0.00,90.00,0,"
  [1351] = "0.00,0.00,0.00,90.00,0.00,90.00,1,"
  [1352] = "0.00,0.00,0.00,90.00,0.00,90.00,0,"
  [1353] = "0.00,0.00,0.00,90.00,0.00,90.00,0,"
  [1354] = "0.00,0.00,0.00,90.00,0.00,90.00,0,"
  [1355] = "0.00,0.00,0.00,90.00,0.00,90.00,1,"
  [1356] = "0.00,0.00,0.00,90.00,0.00,90.00,0,"
  [1357] = "0.00,0.00,0.00,90.00,0.00,90.00,0,"
  [1358] = "0.00,0.00,0.00,90.00,0.00,90.00,0,"
  [1359] = "0.00,0.00,0.00,90.00,0.00,90.00,1,"
  [1360] = "0.00,0.00,0.00,90.00,0.00,90.00,0,"
  [1361] = "0.00,0.00,0.00,90.00,0.00,90.00,0,"
  [1362] = "0.00,0.00,0.00,90.00,0.00,90.00,0,"
  [1363] = "0.00,0.00,0.00,90.00,0.00,90.00,1,"
  [1364] = "0.00,0.00,0.00,90.00,0.00,90.00,0,"
  [1365] = "0.00,0.00,0.00,90.00,0.00,90.00,0,"
  [1366] = "0.00,0.00,0.00,90.00,0.00,90.00,0,"
  [1367] = "0.00,0.00,0.00,90.00,0.00,90.00,1,"
  [1368] = "0.00,0.00,0.00,90.00,0.00,90.00,0,"
  [1369] = "0.00,0.00,0.00,90.00,0.00,90.00,0,"
  [1370] = "0.00,0.00,0.00,90.00,0.00,90.00,0,"
  [1371] = "0.00,0.00,0.00,90.00,0.00,90.00,1,"
  [1372] = "0.00,0.00,0.00,90.00,0.00,90.00,0,"
  [1373] = "0.00,0.00,0.00,90.00,0.00,90.00,0,"
  [1374] = "0.00,0.00,0.00,90.00,0.00,90.00,0,"
  [1375] = "0.00,0.00,0.00,90.00,0.00,90.00,1,"
  [1376] = "0.00,0.00,0.00,90.00,0.00,90.00,0,"
  [1377] = "0.00,0.00,0.00,90.00,0.00,90.00,0,"
  [1378] = "0.00,0.00,0.00,90.00,0.00,90.00,0,"
  [1379] = "0.00,0.00,0.00,90.00,0.00,90.00,1,"
  [1380] = "0.00,0.00,0.00,90.00,0.00,90.00,0,"
  [1381] = "0.00,0.00,0.00,90.00,0.00,90.00,0,"
  [1382] = "0.00,0.00,0.00,90.00,0.00,90.00,0,"
  [1383] = "0.00,0.00,0.00,90.00,0.00,90.00,1,"
  [1384] = "0.00,0.00,0.00,90.00,0.00,90.00,0,"
  [1385] = "0.00,0.00,0.00,90.00,0.00,90.00,0,"
  [1386] = "0.00,0.00,0.00,90.00,0.00,90.00,0,"
  [1387] = "0.00,0.00,0.00,90.00,0.00,90.00,1,"
  [1388] = "0.00,0.00,0.00,90.00,0.00,90.00,0,"
  [1389] = "0.00,0.00,0.00,90.00,0.00,90.00,0,"
  [1390] = "0.00,0.00,0.00,90.00,0.00,90.00,0,"
  [1391] = "0.00,0.00,0.00,90.00,0.00,90.00,1,"
  [1392] = "0.00,0.00,0.00,90.00,0.00,90.00,0,"
  [1393] = "0.00,0.00,0.00,90.00,0.00,90.00,0,"
  [1394] = "0.00,0.00,0.00,90.00,0.00,90.00,0,"
  [1395] = "0.00,0.00,0.00,90.00,0.00,90.00,1,"
  [1396] = "0.00,0.00,0.00,90.00,0.00,90.00,0,"
  [1397] = "0.00,0.00,0.00,90.00,0.00,90.00,0,"
  [1398] = "0.00,0.00,0.00,90.00,0.00,90.00,0,"
  [1399] = "0.00,0.00,0.00,90.00,0.00,90.00,1,"
  [1400] = "0.00,0.00,0.00,90.00,0.00,90.00,0,"
  [1401] = "0.00,0.00,0.00,90.00,0.00,90.00,0,"
  [1402] = "0.00,0.00,0.00,90.00,0.00,90.00,0,"
  [1403] = "0.00,0.00,0.00,90.00,0.00,90.00,1,"
  [1404] = "0.00,0.00,0.00,90.00,0.00,90.00,0,"
  [1405] = "0.00,0.00,0.00,90.00,0.00,90.00,0,"
  [1406] = "0.00,0.00,0.00,90.00,0.00,90.00,0,"
  [1407] = "0.00,0.00,0.00,90.00,0.00,90.00,1,"
  [1408] = "0.00,0.00,0.00,90.00,0.00,90.00,0,"
  [1409] = "0.00,0.00,0.00,90.00,0.00,90.00,0,"
  [1410] = "0.00,0.00,0.00,90.00,0.00,90.00,0,"
  [1411] = "0.00,0.00,0.00,90.00,0.00,90.00,1,"
  [1412] = "0.00,0.00,0.00,90.00,0.00,90.00,0,"
  [1413] = "0.00,0.00,0.00,90.00,0.00,90.00,0,"
  [1414] = "0.00,0.00,0.00,90.00,0.00,90.00,0,"
  [1415] = "0.00,0.00,0.00,90.00,0.00,90.00,1,"
  [1416] = "0.00,0.00,0.00,90.00,0.00,90.00,0,"
  [1417] = "0.00,0.00,0.00,90.00,0.00,90.00,0,"
  [1418] = "0.00,0.00,0.00,90.00,0.00,90.00,0,"
  [1419] = "0.00,0.00,0.00,90.00,0.00,90.00,1,"
  [1420] = "0.00,0.00,0.00,90.00,0.00,90.00,0,"
  [1421] = "0.00,0.00,0.00,90.00,0.00,90.00,0,"
  [1422] = "0.00,0.00,0.00,90.00,0.00,90.00,0,"
  [1423] = "0.00,0.00,0.00,90.00,0.00,90.00,1,"
  [1424] = "0.00,0.00,0.00,90.00,0.00,90.00,0,"
  [1425] = "0.00,0.00,0.00,90.00,0.00,90.00,0,"
  [1426] = "0.00,0.00,0.00,90.00,0.00,90.00,0,"
  [1427] = "0.00,0.00,0.00,90.00,0.00,90.00,1,"
  [1428] = "0.00,0.00,0.00,90.00,0.00,90.00,0,"
  [1429] = "0.00,0.00,0.00,90.00,0.00,90.00,0,"
  [1430] = "0.00,0.00,0.00,90.00,0.00,90.00,0,"
  [1431] = "0.00,0.00,0.00,90.00,0.00,90.00,1,"
  [1432] = "0.00,0.00,0.00,90.00,0.00,90.00,0,"
  [1433] = "0.00,0.00,0.00,90.00,0.00,90.00,0,"
  [1434] = "0.00,0.00,0.00,90.00,0.00,90.00,0,"
  [1435] = "0.00,0.00,0.00,90.00,0.00,90.00,1,"
  [1436] = "0.00,0.00,0.00,90.00,0.00,90.00,0,"
  [1437] = "0.00,0.00,0.00,90.00,0.00,90.00,0,"
  [1438] = "0.00,0.00,0.00,90.00,0.00,90.00,0,"
  [1439] = "0.00,0.00,0.00,90.00,0.00,90.00,1,"
  [1440] = "0.00,0.00,0.00,90.00,0.00,90.00,0,"
  [1441] = "0.00,0.00,0.00,90.00,0.00,90.00,0,"
  [1442] = "0.00,0.00,0.00,90.00,0.00,90.00,0,"
  [1443] = "0.00,0.00,0.00,90.00,0.00,90.00,1,"
  [1444] = "0.00,0.00,0.00,90.00,0.00,90.00,0,"
  [1445] = "0.00,0.00,0.00,90.00,0.00,90.00,0,"
  [1446] = "0.00,0.00,0.00,90.00,0.00,90.00,0,"
  [1447] = "0.00,0.00,0.00,90.00,0.00,90.00,1,"
  [1448] = "0.00,0.00,0.00,90.00,0.00,90.00,0,"
  [1449] = "0.00,0.00,0.00,90.00,0.00,90.00,0,"
  [1450] = "0.00,0.00,0.00,90.00,0.00,90.00,0,"
  [1451] = "0.00,0.00,0.00,90.00,0.00,90.00,1,"
  [1452] = "0.00,0.00,0.00,90.00,0.00,90.00,0,"
  [1453] = "0.00,0.00,0.00,90.00,0.00,90.00,0,"
  [1454] = "0.00,0.00,0.00,90.00,0.00,90.00,0,"
  [1455] = "0.00,0.00,0.00,90.00,0.00,90.00,1,"
  [1456] = "0.00,0.00,0.00,90.00,0.00,90.00,0,"
  [1457] = "0.00,0.00,0.00,90.00,0.00,90.00,0,"
  [1458] = "0.00,0.00,0.00,90.00,0.00,90.00,0,"
  [1459] = "0.00,0.00,0.00,90.00,0.00,90.00,1,"
  [1460] = "0.00,0.00,0.00,90.00,0.00,90.00,0,"
  [1461] = "0.00,0.00,0.00,90.00,0.00,90.00,0,"
  [1462] = "0.00,0.00,0.00,90.00,0.00,90.00,0,"
  [1463] = "0.00,0.00,0.00,90.00,0.00,90.00,1,"
  [1464] = "0.00,0.00,0.00,90.00,0.00,90.00,0,"
  [1465] = "0.00,0.00,0.00,90.00,0.00,90.00,0,"
  [1466] = "0.00,0.00,0.00,90.00,0.00,90.00,0,"
  [1467] = "0.00,0.00,0.00,90.00,0.00,90.00,1,"
  [1468] = "0.00,0.00,0.00,90.00,0.00,90.00,0,"
  [1469] = "0.00,0.00,0.00,90.00,0.00,90.00,0,"
  [1470] = "0.00,0.00,0.00,90.00,0.00,90.00,0,"
  [1471] = "0.00,0.00,0.00,90.00,0.00,90.00,1,"
  [1472] = "0.00,0.00,0.00,90.00,0.00,90.00,0,"
  [1473] = "0.00,0.00,0.00,90.00,0.00,90.00,0,"
  [1474] = "0.00,0.00,0.00,90.00,0.00,90.00,0,"
  [1475] = "0.00,0.00,0.00,90.00,0.00,90.00,1,"
  [1476] = "0.00,0.00,0.00,90.00,0.00,90.00,0,"
  [1477] = "0.00,0.00,0.00,90.00,0.00,90.00,0,"
  [1478] = "0.00,0.00,0.00,90.00,0.00,90.00,0,"
  [1479] = "0.00,0.00,0.00,90.00,0.00,90.00,1,"
  [1480] = "0.00,0.00,0.00,90.00,0.00,90.00,0,"
  [1481] = "0.00,0.00,0.00,90.00,0.00,90.00,0,"
  [1482] = "0.00,0.00,0.00,90.00,0.00,90.00,0,"
  [1483] = "0.00,0.00,0.00,90.00,0.00,90.00,1,"
  [1484] = "0.00,0.00,0.00,90.00,0.00,90.00,0,"
  [1485] = "0.00,0.00,0.00,90.00,0.00,90.00,0,"
  [1486] = "0.00,0.00,0.00,90.00,0.00,90.00,0,"
  [1487] = "0.00,0.00,0.00,90.00,0.00,90.00,1,"
  [1488] = "0.00,0.00,0.00,90.00,0.00,90.00,0,"
  [1489] = "0.00,0.00,0.00,90.00,0.00,90.00,0,"
  [1490] = "0.00,0.00,0.00,90.00,0.00,90.00,0,"
  [1491] = "0.00,0.00,0.00,90.00,0.00,90.00,1,"
  [1492] = "0.00,0.00,0.00,90.00,0.00,90.00,0,"
  [1493] = "0.00,0.00,0.00,90.00,0.00,90.00,0,"
  [1494] = "0.00,0.00,0.00,90.00,0.00,90.00,0,"
  [1495] = "0.00,0.00,0.00,90.00,0.00,90.00,1,"
  [1496] = "0.00,0.00,0.00,90.00,0.00,90.00,0,"
  [1497] = "0.00,0.00,0.00,90.00,0.00,90.00,0,"
  [1498] = "0.00,0.00,0.00,90.00,0.00,90.00,0,"
  [1499] = "0.00,0.00,0.00,90.00,0.00,90.00,1,"
string strCmd = "RBREDY"
string strScrMsg[8]
  [0] = "F1===>robot1 home or ready"
  [1] = "F2===>robot2 home or ready"
  [2] = "F3===>delete points"
  [3] = "F4===>stop sychron"
  [4] = "F5===>start sychron"
  [5] = "F8===>read txt "
tool tTip = {z=66.95, fatherId=flange[0], ioLink=valve1}
public tool tTool = {z=180, fatherId=flange[0], ioLink=valve1}
trsf trsf_test
